// TIA Portal project "bon_nuoc" (V17)

(* hardware
DEVICE "PC-System_1"  SIMATIC PC station
   slot 0: "SIMATIC PC station"  Rail  SIMATIC PC-Station  V1.0
      slot 125: "Stationmanager"  Station_Manager  V6.0.4
   slot 1: "HMI_RT_1"  WinCC RT Advanced  6AV2 104-0xxxx-xxxx  17.0.0.0
      slot 33792: "Computer interface"  Host interface
   slot 2: "IE general_1"  IE General  IE_CP  V8.2.0
      slot 1: "PROFINET interface"  IEGeneral.Interface.8.2.0
DEVICE "S7-1200 station_1"  S7-1200 Station
   slot 0: "Rack_0"  S7-1200 Rack  Rack  V1.0
   slot 1: "PLC_1"  CPU 1214C DC/DC/DC  6ES7 214-1AG40-0XB0  V4.5
*)

// ===== PLC "PLC_1"  CPU 1214C DC/DC/DC =====

VAR_GLOBAL   // PLC tag table "Default tag table"
   "System_Byte" AT %MB1 : Byte;
   "FirstScan" AT %M1.0 : Bool;
   "DiagStatusUpdate" AT %M1.1 : Bool;
   "AlwaysTRUE" AT %M1.2 : Bool;
   "AlwaysFALSE" AT %M1.3 : Bool;
   "Clock_Byte" AT %MB0 : Byte;
   "Clock_10Hz" AT %M0.0 : Bool;
   "Clock_5Hz" AT %M0.1 : Bool;
   "Clock_2.5Hz" AT %M0.2 : Bool;
   "Clock_2Hz" AT %M0.3 : Bool;
   "Clock_1.25Hz" AT %M0.4 : Bool;
   "Clock_1Hz" AT %M0.5 : Bool;
   "Clock_0.625Hz" AT %M0.6 : Bool;
   "Clock_0.5Hz" AT %M0.7 : Bool;
   "PUMP" AT %Q0.0 : Bool;
   "VALVE" AT %Q0.1 : Bool;
END_VAR

DATA_BLOCK "DB"   // DB1
{ S7_Optimized_Access := 'FALSE' }
VERSION : 0.1
   VAR
      "AUTO-MAN" : Bool;
      "START-AUTO" : Bool;
      "STOP-AUTO" : Bool;
      AUTO : Bool;
      "PUMP-AUTO" : Bool;
      "VALVE-AUTO" : Bool;
      "S1-H" : Bool;
      "S2-L" : Bool;
      TG1 : Bool;
      "PV-T1" : DInt;
      "PV-T2" : DInt;
      "START-MAN-PUMP" : Bool;
      "STOP-MAN-PUMP" : Bool;
      "PUMP-MAN" : Bool;
      "START-MAN-VALVE" : Bool;
      "STOP-MAN-VALVE" : Bool;
      "VALVE-MAN" : Bool;
      LEVEL : DInt;
   END_VAR
BEGIN
END_DATA_BLOCK

// folder: System blocks/Program resources

DATA_BLOCK "T1"   // DB2
{ S7_Optimized_Access := 'TRUE' }
AUTHOR : Simatic
FAMILY : IEC
NAME : IEC_TMR
VERSION : 1.0
// stored: InstanceOfName IEC_TIMER
"IEC_TIMER"
BEGIN
END_DATA_BLOCK

DATA_BLOCK "T2"   // DB4
{ S7_Optimized_Access := 'TRUE' }
AUTHOR : Simatic
FAMILY : IEC
NAME : IEC_TMR
VERSION : 1.0
// stored: InstanceOfName IEC_TIMER
"IEC_TIMER"
BEGIN
END_DATA_BLOCK

DATA_BLOCK "IEC_Counter_0_DB"   // DB5
{ S7_Optimized_Access := 'TRUE' }
AUTHOR : Simatic
FAMILY : IEC
NAME : CNTR
VERSION : 1.0
// stored: InstanceOfName IEC_COUNTER
"IEC_COUNTER"
BEGIN
END_DATA_BLOCK

// folder: (top level)

FUNCTION "AUTO" : Void   // FC1, LAD
{ S7_Optimized_Access := 'TRUE' }
VERSION : 0.1
   VAR_TEMP   // added for the SCL form of the ladder/FBD networks
      _w1 : Bool;
   END_VAR
BEGIN

REGION Network 1
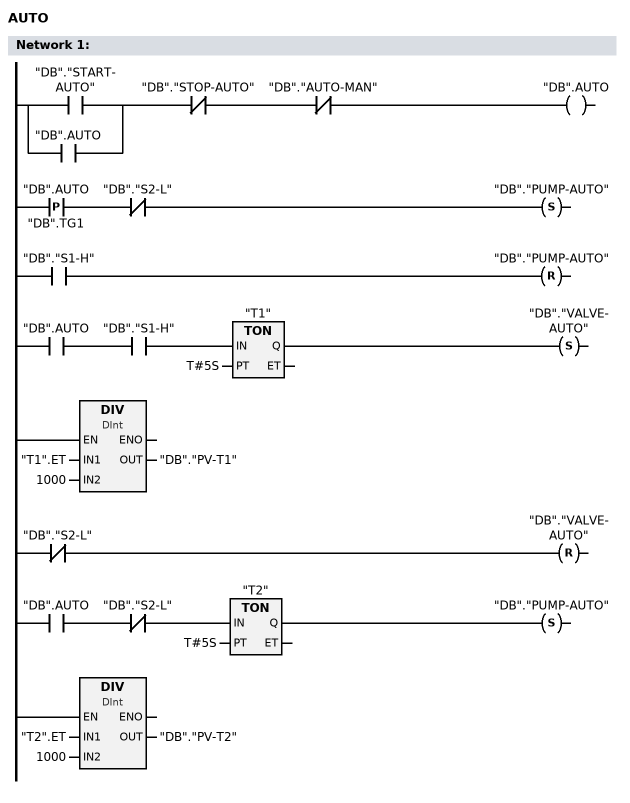
   "DB".AUTO := ("DB"."START-AUTO" OR "DB".AUTO) AND NOT "DB"."STOP-AUTO" AND NOT "DB"."AUTO-MAN";
   #_w1 := "DB".AUTO AND NOT "DB".TG1;   // rising edge of "DB".AUTO
   "DB".TG1 := "DB".AUTO;
   IF #_w1 AND NOT "DB"."S2-L" THEN "DB"."PUMP-AUTO" := TRUE; END_IF;
   IF "DB"."S1-H" THEN "DB"."PUMP-AUTO" := FALSE; END_IF;
   "T1".TON(IN := "DB".AUTO AND "DB"."S1-H", PT := T#5S);
   IF "T1".Q THEN "DB"."VALVE-AUTO" := TRUE; END_IF;
   "DB"."PV-T1" := "T1".ET / 1000;
   IF NOT "DB"."S2-L" THEN "DB"."VALVE-AUTO" := FALSE; END_IF;
   "T2".TON(IN := "DB".AUTO AND NOT "DB"."S2-L", PT := T#5S);
   IF "T2".Q THEN "DB"."PUMP-AUTO" := TRUE; END_IF;
   "DB"."PV-T2" := "T2".ET / 1000;
END_REGION
END_FUNCTION

FUNCTION "MAN" : Void   // FC2, LAD
{ S7_Optimized_Access := 'TRUE' }
VERSION : 0.1
BEGIN

REGION Network 1
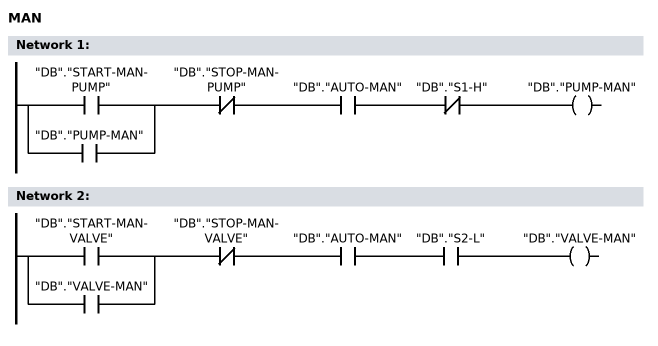
   RUNG wire#powerrail
      Contact( "DB"."START-MAN-PUMP" )
      wire#w1
      I_Contact( "DB"."STOP-MAN-PUMP" )
      Contact( "DB"."AUTO-MAN" )
      I_Contact( "DB"."S1-H" )
      Coil( "DB"."PUMP-MAN" )
   END_RUNG
   RUNG wire#powerrail
      Contact( "DB"."PUMP-MAN" )
   END_RUNG wire#w1
   // the same network as SCL:
   "DB"."PUMP-MAN" := ("DB"."START-MAN-PUMP" OR "DB"."PUMP-MAN") AND NOT "DB"."STOP-MAN-PUMP" AND "DB"."AUTO-MAN" AND NOT "DB"."S1-H";
END_REGION

REGION Network 2
   RUNG wire#powerrail
      Contact( "DB"."START-MAN-VALVE" )
      wire#w1
      I_Contact( "DB"."STOP-MAN-VALVE" )
      Contact( "DB"."AUTO-MAN" )
      Contact( "DB"."S2-L" )
      Coil( "DB"."VALVE-MAN" )
   END_RUNG
   RUNG wire#powerrail
      Contact( "DB"."VALVE-MAN" )
   END_RUNG wire#w1
   // the same network as SCL:
   "DB"."VALVE-MAN" := ("DB"."START-MAN-VALVE" OR "DB"."VALVE-MAN") AND NOT "DB"."STOP-MAN-VALVE" AND "DB"."AUTO-MAN" AND "DB"."S2-L";
END_REGION
END_FUNCTION

FUNCTION "MAP OUTPUT" : Void   // FC3, LAD
{ S7_Optimized_Access := 'TRUE' }
VERSION : 0.1
BEGIN

REGION Network 1
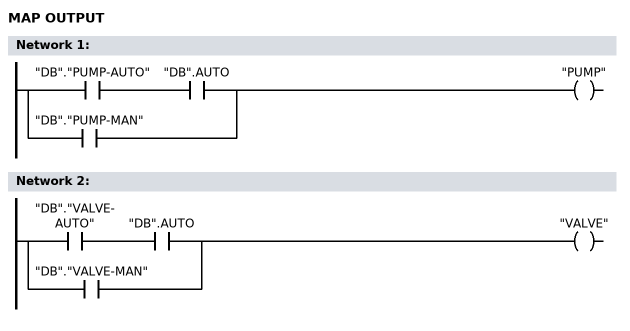
   RUNG wire#powerrail
      Contact( "DB"."PUMP-AUTO" )
      Contact( "DB".AUTO )
      wire#w1
      Coil( "PUMP" )
   END_RUNG
   RUNG wire#powerrail
      Contact( "DB"."PUMP-MAN" )
   END_RUNG wire#w1
   // the same network as SCL:
   "PUMP" := ("DB"."PUMP-AUTO" AND "DB".AUTO) OR "DB"."PUMP-MAN";
END_REGION

REGION Network 2
   RUNG wire#powerrail
      Contact( "DB"."VALVE-AUTO" )
      Contact( "DB".AUTO )
      wire#w1
      Coil( "VALVE" )
   END_RUNG
   RUNG wire#powerrail
      Contact( "DB"."VALVE-MAN" )
   END_RUNG wire#w1
   // the same network as SCL:
   "VALVE" := ("DB"."VALVE-AUTO" AND "DB".AUTO) OR "DB"."VALVE-MAN";
END_REGION
END_FUNCTION

FUNCTION "CHUYEN DONG HMI" : Void   // FC4, LAD
{ S7_Optimized_Access := 'TRUE' }
VERSION : 0.1
BEGIN

REGION Network 1
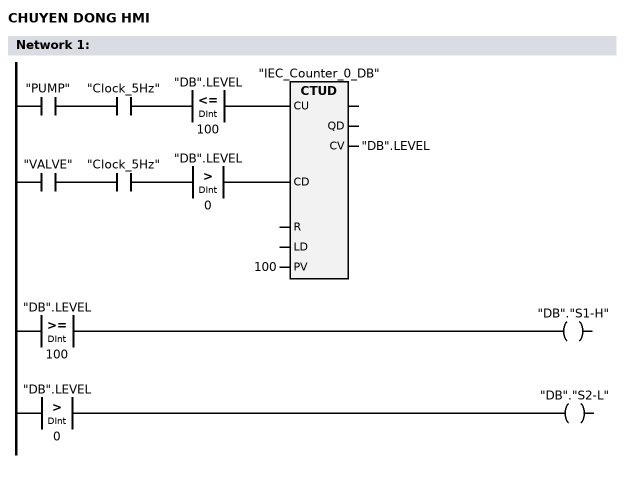
   "IEC_Counter_0_DB".CTUD(CU := "PUMP" AND "Clock_5Hz" AND ("DB".LEVEL <= 100),
                           CD := "VALVE" AND "Clock_5Hz" AND ("DB".LEVEL > 0),
                           PV := 100,
                           CV => "DB".LEVEL);
   "DB"."S1-H" := "DB".LEVEL >= 100;
   "DB"."S2-L" := "DB".LEVEL > 0;
END_REGION
END_FUNCTION

ORGANIZATION_BLOCK "Main"   // OB1, LAD, ProgramCycle
TITLE = "Main Program Sweep (Cycle)"
{ S7_Optimized_Access := 'TRUE' }
VERSION : 0.1
   VAR_INPUT
      Initial_Call : Bool;   // Initial call of this OB
      Remanence : Bool;   // =True, if remanent data are available
   END_VAR
BEGIN

REGION Network 1
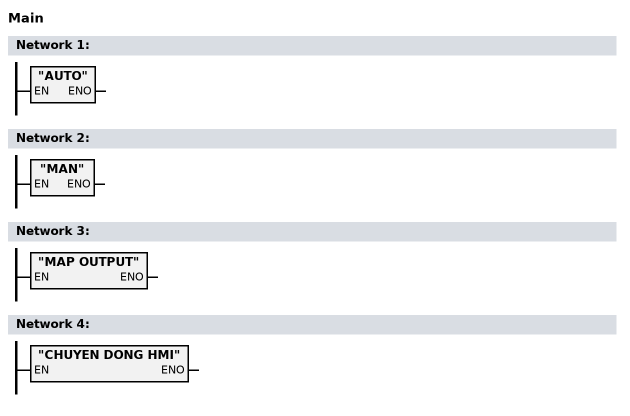
   RUNG wire#powerrail
      "AUTO"()
   END_RUNG
   // the same network as SCL:
   "AUTO"();
END_REGION

REGION Network 2
   RUNG wire#powerrail
      "MAN"()
   END_RUNG
   // the same network as SCL:
   "MAN"();
END_REGION

REGION Network 3
   RUNG wire#powerrail
      "MAP OUTPUT"()
   END_RUNG
   // the same network as SCL:
   "MAP OUTPUT"();
END_REGION

REGION Network 4
   RUNG wire#powerrail
      "CHUYEN DONG HMI"()
   END_RUNG
   // the same network as SCL:
   "CHUYEN DONG HMI"();
END_REGION
END_ORGANIZATION_BLOCK

(* ===== HMI "HMI_RT_1" =====
system functions are stored by id; their names below are inferred from use
connection "HMI_Connection_1": ETHERNET, S7_1200_OMS

HMI tags "Default tag table"
   "DB_AUTO-MAN" : Bool = PLC "DB".AUTO-MAN AT %DB1.DBX0.0, 1 s
   "DB_AUTO" : Bool = PLC "DB".AUTO AT %DB1.DBX0.3, 1 s
   "DB_START-AUTO" : Bool = PLC "DB".START-AUTO AT %DB1.DBX0.1, 1 s
   "DB_STOP-AUTO" : Bool = PLC "DB".STOP-AUTO AT %DB1.DBX0.2, 1 s
   "PUMP" : Bool = PLC PUMP AT %Q0.0, 1 s
   "DB_LEVEL" : DInt = PLC "DB".LEVEL AT %DB1.DBD12, 1 s
   "VALVE" : Bool = PLC VALVE AT %Q0.1, 1 s
   "DB_S1-H" : Bool = PLC "DB".S1-H AT %DB1.DBX0.6, 1 s
   "DB_S2-L" : Bool = PLC "DB".S2-L AT %DB1.DBX0.7, 1 s
   "DB_PV-T1" : DInt = PLC "DB".PV-T1 AT %DB1.DBD2, 1 s
   "DB_PV-T2" : DInt = PLC "DB".PV-T2 AT %DB1.DBD6, 1 s
   "DB_START-MAN-PUMP" : Bool = PLC "DB".START-MAN-PUMP AT %DB1.DBX10.0, 1 s
   "DB_STOP-MAN-PUMP" : Bool = PLC "DB".STOP-MAN-PUMP AT %DB1.DBX10.1, 1 s
   "DB_START-MAN-VALVE" : Bool = PLC "DB".START-MAN-VALVE AT %DB1.DBX10.3, 1 s
   "DB_STOP-MAN-VALVE" : Bool = PLC "DB".STOP-MAN-VALVE AT %DB1.DBX10.4, 1 s

screen "Screen_1" 1024x768
   TextField "Text field_1" at 65,73 size 111x22; Text 'CHON CHE DO'
   Button "Button_1" at 86,152 size 96x32; TextOff 'CHON'
      on Click: InvertBit("DB_AUTO-MAN")
   TextField "Text field_2" at 71,108 size 47x22; Text 'AUTO'
      Appearance <- "DB_AUTO-MAN"
   Circle "Circle_1" at 51,113 size 18x18
      Appearance <- "DB_AUTO-MAN"
   TextField "Text field_3" at 151,108 size 40x22; Text 'MAN'
      Appearance <- "DB_AUTO-MAN"
   Circle "Circle_2" at 131,113 size 18x18
      Appearance <- "DB_AUTO-MAN"
   TextField "Text field_4" at 99,254 size 47x22; Text 'AUTO'
   Circle "Circle_4" at 97,285 size 48x48
      Appearance <- "DB_AUTO"
   Button "Button_2" at 69,346 size 96x32; TextOff 'START'
      on Press: SetBit("DB_START-AUTO")
      on Release: ResetBit("DB_START-AUTO")
   Button "Button_3" at 71,393 size 96x32; TextOff 'STOP'
      on Release: ResetBit("DB_STOP-AUTO")
      on Press: SetBit("DB_STOP-AUTO")
   SymbolLibrary "Symbol library_1" at 330,521 size 266x69
      Appearance <- "PUMP"
      on Activate: function_f294b399("PUMP", 350, 521, 200, 200, -1, -1, 1)
   SymbolLibrary "Symbol library_2" at 629,225 size 151x256
   Slider "Slider_1" at 634,228 size 149x207; Caption 'SIMATIC'
      ProcessValue <- "DB_LEVEL"
   SymbolLibrary "Symbol library_4" at 407,168 size 254x30
   SymbolLibrary "Symbol library_5" at 655,168 size 57x60
   SymbolLibrary "Symbol library_6" at 358,168 size 49x73
   SymbolLibrary "Symbol library_7" at 358,241 size 25x276
   SymbolLibrary "Symbol library_8" at 682,435 size 37x314
   SymbolLibrary "Symbol library_9" at 753,526 size 120x120
   SymbolLibrary "Symbol library_10" at 192,484 size 120x120
   TextField "Text field_5" at 213,534 size 59x22; Text 'WATER'
   SymbolLibrary "Symbol library_3" at 674,528 size 74x120
      Appearance <- "VALVE"
      on Activate: function_efd93a16("VALVE", 750, 400, -1, -1, 1)
   TextField "Text field_6" at 804,541 size 22x59; Text 'WATER'
   SymbolLibrary "Symbol library_11" at 783,225 size 75x29
      Appearance <- "DB_S1-H"
   SymbolLibrary "Symbol library_12" at 785,411 size 75x29
      Appearance <- "DB_S2-L"
   TextField "Text field_7" at 866,224 size 25x22; Text 'S1'
   TextField "Text field_8" at 866,415 size 25x22; Text 'S2'
   IOField "I/O field_1" at 470,279 size 96x32; FormatPattern 9999999999
      ProcessValue <- "DB_PV-T1"
   IOField "I/O field_2" at 471,324 size 96x32; FormatPattern 9999999999
      ProcessValue <- "DB_PV-T2"
   TextField "Text field_9" at 427,285 size 24x22; Text 'T1'
   TextField "Text field_10" at 426,327 size 24x22; Text 'T2'

PopupScreen "VALVE" 240x240
   TextField "Text field_4" at 88,23 size 53x22; Text 'VALVE'
   Button "Button_2" at 66,89 size 96x32; TextOff 'START'
      on Release: ResetBit("DB_START-MAN-VALVE")
      on Press: SetBit("DB_START-MAN-VALVE")
   Button "Button_3" at 66,161 size 96x32; TextOff 'STOP'
      on Release: ResetBit("DB_STOP-MAN-VALVE")
      on Press: SetBit("DB_STOP-MAN-VALVE")

PopupScreen "PUMP" 240x240
   TextField "Text field_4" at 88,23 size 49x22; Text 'PUMP'
   Button "Button_2" at 66,89 size 96x32; TextOff 'START'
      on Release: ResetBit("DB_START-MAN-PUMP")
      on Press: SetBit("DB_START-MAN-PUMP")
   Button "Button_3" at 66,161 size 96x32; TextOff 'STOP'
      on Release: ResetBit("DB_STOP-MAN-PUMP")
      on Press: SetBit("DB_STOP-MAN-PUMP")
*)